// TIA Portal V17 export
FUNCTION "并联_多支路" : Void   // FC, LAD
{ S7_Optimized_Access := 'TRUE' }
VERSION : 0.1
// stored: AutoNumber true, IsIECCheckEnabled false, SetENOAutomatically false
BEGIN

REGION Network 1
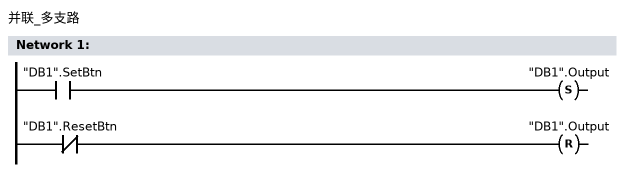
   RUNG wire#powerrail
      Contact( "DB1".SetBtn )
      S_Coil( "DB1".Output )
   END_RUNG
   RUNG wire#powerrail
      I_Contact( "DB1".ResetBtn )
      R_Coil( "DB1".Output )
   END_RUNG
   // the same network as SCL:
   IF "DB1".SetBtn THEN "DB1".Output := TRUE; END_IF;
   IF NOT "DB1".ResetBtn THEN "DB1".Output := FALSE; END_IF;
END_REGION
END_FUNCTION
